Fanuc KAREL source: ko00019.KL

PROGRAM KO00019
%STACKSIZE=65535
%PRIORITY=65535
%NOLOCKGROUP
VAR
P1 : XYZWPREXT
P2 : XYZWPREXT
P3 : XYZWPREXT
OUT : XYZWPREXT
BEGIN
-- UNRESOLVED_PC line 9 opcodes [27 27 49 7E AD 27 49 7E AD 27 49 7E AD 76 7E 4A] marker_code=0
END KO00019
